FUNCTION projArray1 : BOOL
VAR_INPUT
	arr: ARRAY[0..2] OF BOOL;
	idx: DINT;
END_VAR

projArray1 := arr[normProjIdx(idx, 3)];

END_FUNCTION

(* stored: Version 1.1.0.1, ProductVersion 3.1.4022.18
   POU projArray1: Id {14389202-a35a-4b98-bc7b-f8cefed4c7ce}, SpecialFunc None *)
